{attribute 'qualified_only'}
{attribute 'strict'}
TYPE MsgLevel :
(
	Error	:= 4,
	Alarm	:= 2,
	Info	:= 1,
	None	:= 0
	
)INT;
END_TYPE

(* stored: Version 1.1.0.1, ProductVersion 3.1.4024.14
   DUT MsgLevel: Id {dd05dac5-7205-4b5c-97dc-5995ff810108} *)
